KUKA KRL program: PolishMain01.src, PolishMain01.dat

--- PolishMain01.src ---
&ACCESS RVP
&REL 133
&COMMENT Polish 250608
&PARAM DISKPATH = KRC:\R1\Program\SbtComm012Polish
def  PolishMain01 ( )
;FOLD INI;%{PE}
  ;FOLD BASISTECH INI
    GLOBAL INTERRUPT DECL 3 WHEN $STOPMESS==TRUE DO IR_STOPM ( )
    INTERRUPT ON 3
    BAS (#INITMOV,0 )
  ;ENDFOLD (BASISTECH INI)
  ;FOLD USER INI
    ;Make your modifications here

  ;ENDFOLD (USER INI)
;ENDFOLD (INI)
;Initialized Data
PolishInitialization()
;FOLD SbtComm012.PolishInit ;%{PE}
WAIT SEC 0.0
Comm012HeadStatus(1)
Comm012HeadStatus(2)
Comm012HeadStatus(3)
Comm012HeadStatus(4)
Comm012PolishInit()
;ENDFOLD
;Camera photography
PolishTrigger01()
;FOLD SbtComm012.PolishPlanning IN Job Id: 1, IN Planing Id: 1, OUT Num Edges: NumOfPath ;%{PE}
Comm012PolishPlan(1, 1, NumOfPath)
;ENDFOLD
for PathNumber = 1 to NumOfPath
;FOLD SbtComm012.PolishGetParam IN Job Id: 1, IN Num Edges: PathNumber, OUT GrindHead Id: GrindHead, OUT Spindle Speed: SpindleSpeed ;%{PE}
Comm012PolishGetPara(1, PathNumber, GrindHead, SpindleSpeed)
;ENDFOLD
;FOLD Replace the polishing head
;PolishReplaceHead(GrindHead)
;ENDFOLD
BAS(#TOOL, GrindHeadTool[GrindHead].BindToolNum)
;FOLD SbtComm012.PolishGetPath IN Job Id: 1, IN Num Edges: PathNumber, IN Step Dist: 5 ;%{PE}
Comm012PolishGetPath(1,  PathNumber, 5)
;ENDFOLD
;FOLD SbtComm012.HeadCtrlByName IN Ctrl Type: HEAD_STARTING, IN GrindHead Id: GrindHead, IN Spindle Speed: SpindleSpeed, IN Timeout: 0 sec ;%{PE}
WAIT SEC 0.0
Comm012HeadCtrl(#HEAD_STARTING, GrindHead, SpindleSpeed, 0 * 1000)
;ENDFOLD
;FOLD SbtComm012.PolishMoveAppr IN Speed Type: EXTERNAL, IN GrindHead Id: GrindHead, IN Move Speed: 300 cm/min ;%{PE}
IF 1 == 1 THEN
Comm012PolishMoveAppr(GrindHead, )
ELSE
Comm012PolishMoveAppr(GrindHead, 300)
ENDIF
;ENDFOLD
;FOLD SbtComm012.HeadCtrlByName IN Ctrl Type: HEAD_STARTING, IN GrindHead Id: GrindHead, IN Spindle Speed: SpindleSpeed, IN Timeout: 10 sec ;%{PE}
WAIT SEC 0.0
Comm012HeadCtrl(#HEAD_STARTING, GrindHead, SpindleSpeed, 10 * 1000)
;ENDFOLD
;FOLD SbtComm012.PolishMoveGrind IN Speed Type: EXTERNAL, IN GrindHead Id: GrindHead, IN Move Speed: 300 cm/min, IN Ori Type: VAR ;%{PE}
IF 1 == 1 THEN
Comm012PolishMoveGrind(GrindHead, , #VAR)
ELSE
Comm012PolishMoveGrind(GrindHead, 300, #VAR)
ENDIF
;ENDFOLD
;FOLD SbtComm012.PolishMoveExit IN Speed Type: EXTERNAL, IN GrindHead Id: GrindHead, IN Move Speed: 300 cm/min ;%{PE}
IF 1 == 1 THEN
Comm012PolishMoveExit(GrindHead, )
ELSE
Comm012PolishMoveExit(GrindHead, 300)
ENDIF
;ENDFOLD
endfor
;FOLD SbtComm012.HeadCtrlByName IN Ctrl Type: HEAD_STOPPED, IN GrindHead Id: GrindHead, IN Spindle Speed: SpindleSpeed, IN Timeout: 5 sec ;%{PE}
WAIT SEC 0.0
Comm012HeadCtrl(#HEAD_STOPPED, GrindHead, SpindleSpeed, 5 * 1000)
;ENDFOLD

end

--- PolishMain01.dat ---
&ACCESS RVP
&REL 133
&COMMENT Polish 250608
&PARAM DISKPATH = KRC:\R1\Program\SbtComm012Polish
DEFDAT  POLISHMAIN01
;FOLD EXTERNAL DECLARATIONS;%{PE}%MKUKATPBASIS,%CEXT,%VCOMMON,%P
;FOLD BASISTECH EXT;%{PE}%MKUKATPBASIS,%CEXT,%VEXT,%P
EXT  BAS (BAS_COMMAND  :IN,REAL  :IN )
DECL INT SUCCESS
;ENDFOLD (BASISTECH EXT)
;FOLD USER EXT;%{E}%MKUKATPUSER,%CEXT,%VEXT,%P
;Make your modifications here

;ENDFOLD (USER EXT)
;ENDFOLD (EXTERNAL DECLARATIONS)

DECL INT PathNumber
DECL MODULEPARAM_T LAST_TP_PARAMS={PARAMS[] "SBTCOMM012.SLEEPTIME=0.1; SBTCOMM012.CAMERAID=1; SBTCOMM012.POINTID=1; SBTCOMM012.JOBID=1; SBTCOMM012.PLANID=1; SBTCOMM012.NUNOFEDGES=NumOfEdges1; SBTCOMM012.PATHTYPE=1; SBTCOMM012.EDGE=PathNumber; SBTCOMM012.INTERVALDISTANCE=5; SBTCOMM012.NUMOFEDGES=NumOfPath; SBTCOMM012.POLISHHEAD=PolishHead5; SBTCOMM012.SPINDLESPEED=SpindleSpeed; BASIC.OVERRIDESPEED=30; SBTCOMM012.PLANNINGID=1; SBTCOMM012.GRINDHEADIDBYNAME_=GrindHead1; SBTCOMM012.STEPDISTANCE=5; SBTCOMM012.MOVESPEED=300; SBTCOMM012.GRINDHEADIDBYNAME=GrindHead; SBTCOMM012.SPEED=SpindleSpeed; SBTCOMM012.APPSPEEDTYPE=1; SBTCOMM012.ORITYPE=#VAR; SBTCOMM012.SPINDLESPEEDBYNAME=SpindleSpeed; SBTCOMM012.TIMEOUT=0; SBTCOMM012.GRINDENABLE=False; SBTCOMM012.HEADCTRLTYPE=#HEAD_STARTING                                    "}
DECL INT NumOfEdges1=0
DECL INT PolishHead1=0
DECL REAL SpindleSpeed1=0.0
DECL INT ToolNumber1=0

DECL INT NumOfPath=0
DECL INT GrindHead=0
DECL REAL SpindleSpeed=0.0
ENDDAT
